if DEBUG:
    print(f"Holes without solution: {holes_no_solution}")
    debuglist.append(f"Holes without solution: {holes_no_solution}")

    current_time = datetime.datetime.now()
    filename = os.path.splitext(os.path.basename(__file__))
    with open("C:/Users/Laura/Documents/1.Windesheim/Stage/2024/Lectoraat/Deelvragen/2.Targets maken/debugfile.txt", "a") as file:
        file.write("\n\n-----------------------------------------------\n")
        file.write(current_time.strftime("%c"))
        file.write("\n-----------------------------------------------\n")
        for prints in debuglist:
            file.write(prints)
            file.write("\n")
        file.write(holes_no_solution)
        file.write(filename[0])

--- Python program Addmoveshanktoprog ---
from robodk import robolink, robomath

# Connect to RoboDK
RDK = robolink.Robolink()

# Ask the user to select the program to duplicate
orig_prog = RDK.ItemUserPick("Select the program to duplicate", robolink.ITEM_TYPE_PROGRAM)
if not orig_prog.Valid():
    print("No valid program selected.")
    quit()

# Create a new program (a duplicate) with a new name
new_prog_name = "New_" + orig_prog.Name()
new_prog = RDK.AddProgram(new_prog_name)
print("Creating new program:", new_prog.Name())

# Get the number of instructions from the original program
ins_count = orig_prog.InstructionCount()
print("Original program '{}' has {} instructions.".format(orig_prog.Name(), ins_count))

# Iterate over each instruction in the original program
for i in range(ins_count):
    # Retrieve instruction info as a dictionary.
    # Note: Calling setParam(i) with only the index returns the instruction information.
    ins_dict = orig_prog.setParam(i)

    # Try to get the command code string from the instruction dictionary.
    # (Many instructions have a "Code" key that holds the Python command as text.)
    code_line = ins_dict.get("Code", "").strip()
    if not code_line:
        print("Skipping instruction {} because no code is available.".format(i))
        continue

    # Add the instruction to the new program
    print("Adding instruction {}: {}".format(i, code_line))
    new_prog.RunInstruction(code_line, robolink.INSTRUCTION_CALL_PROGRAM)

    # If the instruction contains "FaceTarget" then add two extra moveshank instructions after it.
    if "Face_Target" in code_line:
        print("Detected 'FaceTarget' at instruction {}. Inserting moveshank instructions.".format(i))
        new_prog.RunInstruction('move_shank(20)', robolink.INSTRUCTION_CALL_PROGRAM)
        new_prog.RunInstruction('move_shank(0)', robolink.INSTRUCTION_CALL_PROGRAM)

# Finalize the new program; this applies the modifications
new_prog.Update()
print("New program '{}' created successfully.".format(new_prog.Name()))

--- Python program importerTest ---
# This macro loads CSV target files and places them in RoboDK
# Supported CSV format: X,Y,Z,RX,RY,RZ

# Import required modules
from robodk.robolink import *  # API to communicate with RoboDK
from robodk.robomath import *  # Robot toolbox
from robodk.robodialogs import *
from robodk.robofileio import *
import robodk.robolinkutils as RDKutils

# Start communication with RoboDK
RDK = Robolink()

# Ask the user to select the robot
ROBOT = RDK.ItemUserPick('Select a robot', ITEM_TYPE_ROBOT)

# Check if the user selected a robot
if not ROBOT.Valid():
    quit()

# Get the reference frame and active tool
BASE = ROBOT.Parent()
FRAME = RDK.ItemUserPick('Reference Frame', ITEM_TYPE_FRAME)
FRAMEPOSE = RDKutils.getPoseWrt(FRAME, BASE)  # frame pose wrt robot base
TOOL = ROBOT.getLink(ITEM_TYPE_TOOL)
TOOLPOSE = RDKutils.getPoseWrt(TOOL, TOOL.Parent())  # tool pose wrt robot flange

if not FRAME.Valid() or not TOOL.Valid():
    raise Exception("Select appropriate FRAME and TOOL references")

# Function to convert XYZWPR to a pose
def xyzwpr_to_pose(xyzwpr):
    x, y, z, rx, ry, rz = xyzwpr
    return point_Zaxis_2_pose([x, y, z], [rx, ry, rz])

# Ask user to select the CSV file
csv_file = getOpenFileName(RDK.getParam('PATH_OPENSTATION'))

# Specify file codec
codec = 'utf-8'

# Load CSV target data
def load_targets(strfile):
    csvdata = LoadList(strfile, ',', codec)
    poses = []
    idxs = []
    for i in range(0, len(csvdata)):
        x, y, z, rx, ry, rz = csvdata[i][0:6]
        poses.append(xyzwpr_to_pose([x, y, z, rx, ry, rz]))
        idxs.append(i)
    return poses, idxs

# Create targets in RoboDK and move the robot to each target
def process_targets(strfile):
    poses, idxs = load_targets(strfile)
    program_name = getFileName(strfile)
    program_name = program_name.replace('-', '_').replace(' ', '_')

    # Set the robot's frame and tool
    ROBOT.setFrame(FRAME)
    ROBOT.setTool(TOOL)

    # Create a program to visit all targets
    program = RDK.AddProgram('Visit_' + program_name, ROBOT)

    for pose, idx in zip(poses, idxs):
        # Create target name
        name = 'Target-%s-%i' % (program_name, idx)

        # Delete target if it already exists
        target = RDK.Item(name, ITEM_TYPE_TARGET)
        if target.Valid():
            target.Delete()

        # Create new target
        target = RDK.AddTarget(name, FRAME, ROBOT)
        target.setPose(pose)

        # Add a movement instruction to the program
        program.MoveJ(target)

        # Optional: Move the robot to the target in simulation
        RDK.setSimulationSpeed(1)  # Normal speed
        ROBOT.MoveJ(target)

# Main execution
if __name__ == "__main__":
    # Ask user whether to just create targets or also move the robot
    move_robot = RDK.RunMode() != RUNMODE_SIMULATE

    if move_robot:
        # We're in run mode, just move the robot to targets
        poses, idxs = load_targets(csv_file)
        for pose, idx in zip(poses, idxs):
            ROBOT.MoveJ(pose)
    else:
        # We're in simulation mode, create targets and a program
        process_targets(csv_file)

    RDK.ShowMessage("Target processing complete", False)

--- program Prog20 (robot UR10e) ---
  Set Ref.: CSV Frame
  Set Tool: TCP Schroeftool
  MoveL (Target 36)
  Call Program_Face_-1_0_0
  Call Program_Face_-1_0_0
  MoveL (Target 36)
  MoveL (Target 35)
  MoveJ (Target 37 new)
  MoveL (Target 37 new)
  MoveL (Target 35)
  Call Program_Face_0_-1_1
  MoveL (Target 35)
  Call Program_Face_0_-1_0
  MoveL (Target 35)

--- program Program_Face_-1_0_0 (robot UR10e) ---
  Set Ref.: CSV Frame
  Set Tool: TCP Schroeftool
  MoveL (Target 36)
  MoveL (Face_Target_-1_0_0)
  MoveL (H-12.5_30.0-9)
  MoveL (Face_Target_-1_0_0)
  MoveL (H-12.5_30.0-10)
  MoveL (Face_Target_-1_0_0)
  MoveL (H-12.5_30.0-11)
  MoveL (Face_Target_-1_0_0)
  MoveL (H-12.5_30.0-12)
  MoveL (Face_Target_-1_0_0)
  MoveL (H-12.5_30.0-13)
  MoveL (Face_Target_-1_0_0)
  MoveL (H-12.5_30.0-14)
  MoveL (Face_Target_-1_0_0)
  MoveL (H-12.5_30.0-15)
  MoveL (Face_Target_-1_0_0)
  MoveL (Target 36)

--- program Program_Face_0_0_1 (robot UR10e) ---
  Set Ref.: CSV Frame
  Set Tool: TCP Schroeftool
  MoveL (Face_Target_0_0_1)
  MoveL (H-12.4_20.0-0)
  MoveL (Face_Target_0_0_1)
  MoveL (H-12.4_20.0-1)
  MoveL (Face_Target_0_0_1)
  MoveL (H-12.4_20.0-2)
  MoveL (Face_Target_0_0_1)
  MoveL (H-12.4_20.0-3)
  MoveL (Face_Target_0_0_1)
  MoveL (H-12.4_20.0-4)
  MoveL (Face_Target_0_0_1)
  MoveL (H-12.4_20.0-5)
  MoveL (Face_Target_0_0_1)
  MoveL (H-12.4_20.0-6)
  MoveL (Face_Target_0_0_1)

--- program Program_Face_0_-1_1 (robot UR10e) ---
  Set Ref.: CSV Frame
  Set Tool: TCP Schroeftool
  MoveL (Target 35)
  MoveJ (Target 37 new)
  MoveL (Toolswitch-m8)
  Call move_shank(20)
  Call move_shank(0)
  MoveL (Aanlevering-Pos1)
  Call move_shank(20)
  Call move_shank(0)
  MoveJ (Target 37 new)
  MoveJ (Target 35)
  MoveL (Face_Target_0_-1_1)
  MoveL (H-12.4_20.0-10)
  Call move_shank(20)
  Call move_shank(0)
  MoveL (Target 35)
  MoveJ (Target 37 new)
  MoveL (Aanlevering-Pos1)
  Call move_shank(20)
  Call move_shank(0)
  MoveJ (Target 37 new)
  MoveJ (Target 35)
  MoveL (Face_Target_0_-1_1)
  MoveL (H-12.4_20.0-11)
  Call move_shank(20)
  Call move_shank(0)
  MoveL (Target 35)
  MoveJ (Target 37 new)
  MoveL (Aanlevering-Pos1)
  Call move_shank(20)
  Call move_shank(0)
  MoveJ (Target 37 new)
  MoveJ (Target 35)
  MoveL (Face_Target_0_-1_1)
  MoveL (H-12.4_20.0-12)
  Call move_shank(20)
  Call move_shank(0)
  MoveL (Target 35)
  MoveJ (Target 37 new)
  MoveL (Aanlevering-Pos1)
  Call move_shank(20)
  Call move_shank(0)
  MoveJ (Target 37 new)
  MoveJ (Target 35)
  MoveL (Face_Target_0_-1_1)
  MoveL (H-12.4_20.0-13)
  Call move_shank(20)
  Call move_shank(0)
  MoveL (Target 35)
  MoveJ (Target 37 new)
  MoveL (Aanlevering-Pos1)
  Call move_shank(20)
  Call move_shank(0)
  MoveJ (Target 37 new)
  MoveJ (Target 35)
  MoveL (Face_Target_0_-1_1)
  MoveL (H-12.4_20.0-14)
  Call move_shank(20)
  Call move_shank(0)
  MoveL (Target 35)
  MoveJ (Target 37 new)
  MoveL (Aanlevering-Pos1)
  Call move_shank(20)
  Call move_shank(0)
  MoveJ (Target 37 new)
  MoveL (Target 35)
  - Wanneer face target wordt gemaakt, tussen elke gat moet een helicoil opgepakt worden
- manier bedenken om "Aanlevering-Pos1" target te zoeken 
- manier om Toolswitch-m8 target te zoeken
- wanneer de aanlevering of toolswitch benadert wordt moet dat via target 35 -> target 37

wat er nu aangepast moet worden, moet via de approach points benaderd worden 
de flow voor een gat is de volgende Target 35 -> Target 37 -> Oppakken helicoil, dan via hetzelfde route terug gaan, Target 37 -> Target 35 en naar approach. 
voor elke gat moeten er minimaal 5 bewegingen komen

--- program Program_Face_0_-1_1_m8 (robot UR10e) ---
  Set Ref.: CSV Frame
  Set Tool: TCP Schroeftool
  MoveL (Target 35)
  MoveJ (Target 37 new)
  MoveL (Toolswitch-m8)
  Call move_shank(20)
  Call move_shank(0)
  MoveL (Aanlevering-Pos1)
  Call move_shank(20)
  Call move_shank(0)
  MoveJ (Target 37 new)
  MoveJ (Target 35)
  MoveJ (Target 37 new)
  MoveL (Aanlevering-Pos1)
  Call move_shank(20)
  Call move_shank(0)
  MoveJ (Target 37 new)
  MoveJ (Target 35)
  MoveL (Face_Target_0_-1_1)
  MoveL (H-8.3_20.0-8)
  Call move_shank(20)
  Call move_shank(0)
  MoveL (Target 35)
  MoveJ (Target 37 new)
  MoveL (Aanlevering-Pos1)
  Call move_shank(20)
  Call move_shank(0)
  MoveJ (Target 37 new)
  MoveJ (Target 35)
  MoveL (Face_Target_0_-1_1)
  MoveL (H-8.3_20.0-9)
  Call move_shank(20)
  Call move_shank(0)
  MoveL (Target 35)
  MoveJ (Target 37 new)
  MoveL (Aanlevering-Pos1)
  Call move_shank(20)
  Call move_shank(0)
  MoveJ (Target 37 new)
  MoveJ (Target 35)
  MoveL (Face_Target_0_-1_1)
  MoveL (H-8.3_20.0-10)
  Call move_shank(20)
  Call move_shank(0)
  MoveL (Target 35)
  MoveJ (Target 37 new)
  MoveL (Aanlevering-Pos1)
  Call move_shank(20)
  Call move_shank(0)
  MoveJ (Target 37 new)
  MoveJ (Target 35)
  MoveL (Face_Target_0_-1_1)
  MoveL (H-8.3_20.0-11)
  Call move_shank(20)
  Call move_shank(0)
  MoveL (Target 35)
  MoveJ (Target 37 new)
  MoveL (Aanlevering-Pos1)
  Call move_shank(20)
  Call move_shank(0)
  MoveJ (Target 37 new)
  MoveL (Target 35)
  MoveJ (Target 37 new)
  MoveL (Aanlevering-Pos1)
  Call move_shank(20)
  Call move_shank(0)
  MoveJ (Target 37 new)
  MoveJ (Target 35)
  MoveL (Face_Target_0_-1_1)
  MoveL (H-8.3_20.0-12)
  Call move_shank(20)
  Call move_shank(0)
  MoveL (Target 35)
  MoveJ (Target 37 new)
  MoveL (Aanlevering-Pos1)
  Call move_shank(20)
  Call move_shank(0)
  MoveJ (Target 37 new)
  MoveJ (Target 35)
  MoveL (Face_Target_0_-1_1)
  MoveL (H-8.3_20.0-13)
  Call move_shank(20)
  Call move_shank(0)
  MoveL (Target 35)
  - Wanneer face target wordt gemaakt, tussen elke gat moet een helicoil opgepakt worden
- manier bedenken om "Aanlevering-Pos1" target te zoeken 
- manier om Toolswitch-m8 target te zoeken
- wanneer de aanlevering of toolswitch benadert wordt moet dat via target 35 -> target 37

wat er nu aangepast moet worden, moet via de approach points benaderd worden 
de flow voor een gat is de volgende Target 35 -> Target 37 -> Oppakken helicoil, dan via hetzelfde route terug gaan, Target 37 -> Target 35 en naar approach. 
voor elke gat moeten er minimaal 5 bewegingen komen

--- program Program_Face_0_-1_0 (robot UR10e) ---
  Set Ref.: CSV Frame
  Set Tool: TCP Schroeftool
  MoveL (Face_Target_0_-1_0)
  MoveL (H-12.4_20.0-18)
  MoveL (Face_Target_0_-1_0)
  MoveL (H-12.4_20.0-19)
  MoveL (Face_Target_0_-1_0)
  MoveL (H-12.4_20.0-20)
  MoveL (Face_Target_0_-1_0)
  MoveL (H-12.4_20.0-21)
  MoveL (Face_Target_0_-1_0)
  MoveL (H-12.4_20.0-22)
  MoveL (Face_Target_0_-1_0)

--- program Prog22 (robot UR10e) ---
  Set Ref.: CSV Frame
  Set Tool: TCP Schroeftool
  MoveL (Target 36)
  MoveL (Target 35)
  MoveJ (Target 37 new)
  MoveL (Toolswitch-m8)
  Call move_shank(20)
  Call move_shank(0)
  MoveL (H-10.2_4-0) -> target Aanlevering-Pos1
  Call move_shank(20)
  Call move_shank(0)
  MoveL (Target 37 new)

--- program Visit_8.3_20.0 (robot UR10e) ---
  MoveJ (Target-8.3_20.0-0) [its target is no longer in the station]

--- program Visit_8.3_20.0 (robot UR10e) ---
  MoveJ (Target-8.3_20.0-0) [its target is no longer in the station]
  MoveJ (Target-8.3_20.0-1) [its target is no longer in the station]
  MoveJ (Target-8.3_20.0-2) [its target is no longer in the station]
  MoveJ (Target-8.3_20.0-3) [its target is no longer in the station]
  MoveJ (Target-8.3_20.0-4) [its target is no longer in the station]
  MoveJ (Target-8.3_20.0-5) [its target is no longer in the station]
  MoveJ (Target-8.3_20.0-6) [its target is no longer in the station]
  MoveJ (Target-8.3_20.0-7) [its target is no longer in the station]
  MoveJ (Target-8.3_20.0-8) [its target is no longer in the station]
  MoveJ (Target-8.3_20.0-9) [its target is no longer in the station]
  MoveJ (Target-8.3_20.0-10) [its target is no longer in the station]
  MoveJ (Target-8.3_20.0-11) [its target is no longer in the station]
  MoveJ (Target-8.3_20.0-12) [its target is no longer in the station]
  MoveJ (Target-8.3_20.0-13) [its target is no longer in the station]
  MoveJ (Target-8.3_20.0-14) [its target is no longer in the station]
  MoveJ (Target-8.3_20.0-15) [its target is no longer in the station]

--- program Visit_8.3_20.0 (robot UR10e) ---
  MoveJ (Target-8.3_20.0-0) [its target is no longer in the station]
  MoveJ (Target-8.3_20.0-1) [its target is no longer in the station]
  MoveJ (Target-8.3_20.0-2) [its target is no longer in the station]
  MoveJ (Target-8.3_20.0-3) [its target is no longer in the station]
  MoveJ (Target-8.3_20.0-4) [its target is no longer in the station]
  MoveJ (Target-8.3_20.0-5) [its target is no longer in the station]
  MoveJ (Target-8.3_20.0-6) [its target is no longer in the station]
  MoveJ (Target-8.3_20.0-7) [its target is no longer in the station]
  MoveJ (Target-8.3_20.0-8) [its target is no longer in the station]
  MoveJ (Target-8.3_20.0-9) [its target is no longer in the station]
  MoveJ (Target-8.3_20.0-10) [its target is no longer in the station]
  MoveJ (Target-8.3_20.0-11) [its target is no longer in the station]
  MoveJ (Target-8.3_20.0-12) [its target is no longer in the station]
  MoveJ (Target-8.3_20.0-13) [its target is no longer in the station]
  MoveJ (Target-8.3_20.0-14) [its target is no longer in the station]
  MoveJ (Target-8.3_20.0-15) [its target is no longer in the station]
  MoveJ (Target-8.3_20.0-16) [its target is no longer in the station]
  MoveJ (Target-8.3_20.0-17) [its target is no longer in the station]
  MoveJ (Target-8.3_20.0-18) [its target is no longer in the station]

--- program Prog28 (robot UR10e) ---
  Set Ref.: CSV Frame
  Set Tool: TCP Schroeftool
  MoveL (Target 93)
  MoveL (Target 94)
  MoveL (H-8.3_20.0-0)

--- program Prog29 (robot UR10e) ---
  Set Ref.: CSV Frame
  Set Tool: OnRobot screwdriver kopstuk-inleren
  MoveJ (Target 37 new)
  MoveL (OPPAK)
  Call screw_in(20)
  MoveJ (Target 37 new)
  MoveJ (Target 35)
  MoveL (Face_Target_0_-1_1)
  MoveL (H-8.3_20.0-8)
  Call screw_in(20)
  Call screw_out(20)
  MoveL (Target 35)
  Call Program1
  Call move_shank(0)
  MoveJ (Target 37 new)
  MoveL (OPPAK)
  Call screw_in(20)
  MoveJ (Target 37 new)
  MoveJ (Target 35)
  MoveL (Face_Target_0_-1_1)
  MoveL (H-8.3_20.0-9)
  Call screw_in(20)
  Call screw_out(20)
  MoveL (Target 35)
  Call Program1
  MoveJ (Target 37 new)
  MoveL (OPPAK)
  Call screw_in(20)
  MoveJ (Target 37 new)
  MoveJ (Target 35)
  MoveL (Face_Target_0_-1_1)
  MoveL (H-8.3_20.0-10)
  Call screw_in(20)
  Call screw_out(20)
  MoveL (Target 35)
  Call Program1
